Staubli VAL3: setFrame.pgx

public program setFrame(num nFrame (dimensions=1))
begin
  switch nFrame
    case 0
      frActive=world
    break
    case 1
      frActive=frHotel
    break
    case 2
      frActive=frBeam
    break
    case 3
      frActive=frRack
    break
    default
      logMsg("erro setFrame: "+chr(nFrame))
    break
  endSwitch
end
